// TIA Portal V16 export
// export: Created 2021-07-12T14:47:18.8029087Z, ExportSetting WithDefaults, DisplayName Totally Integrated Automation Portal, DisplayVersion V16, DisplayName TIA Portal Version Control Interface, DisplayVersion V16, DisplayName TIA Portal Openness, DisplayVersion V16, DisplayName STEP 7 Professional, DisplayVersion V16, DisplayName STEP 7 Safety, DisplayVersion V16, DisplayName WinCC Professional, DisplayVersion V16
TYPE "LSimaHydTO_typeInternalMotionData"
TITLE = LSimaHydTO_typeInternalMotionData
// Motion command data
// stored: IsFailsafeCompliant false
   STRUCT
      PositionControlled : Bool := FALSE;   // Activates position controller
      ForceLimited : Bool := FALSE;   // Enable force limiting
      ForceControlled : Bool := FALSE;   // Enable force control
      RampingForward : Bool;   // enable signal for ramping in positive direction
      RampingBackward : Bool;   // enable signal for ramping in negative direction
      ForceCmdTracking { S7_SetPoint := 'True'} : "LSimaHydTO_typeInternalCmdTracking";   // Force command tracking
      DirectOutput { S7_SetPoint := 'True'} : "LSimaHydTO_typeInternalStatusDirectOutput";
   END_STRUCT;
END_TYPE
